FUNCTION_BLOCK FB_Cylinder_DualPWM_DualSensor EXTENDS FB_Cylinder_DualSensor
VAR_INPUT
END_VAR
VAR_OUTPUT
END_VAR
VAR
	fbPWMControl		: FB_Enfield_LSV_PWM_SolenoidControl;
	
	//Internal Property Values
	nDutyCycle		: INT := 100;
	
END_VAR

PROPERTY DutyCycle : INT
GET
DutyCycle := nDutyCycle;
END_GET
SET
nDutyCycle := DutyCycle;
END_SET
END_PROPERTY

METHOD HardwareUpdate : BOOL
VAR_INPUT
END_VAR
SUPER^.HardwareUpdate();

IF bExtendCommand THEN
	fbPWMControl.Actuate(nDutyCycle);
ELSIF bRetractCommand THEN
	fbPWMControl.Actuate(nDutyCycle * -1);
ELSE
	fbPWMControl.Actuate(0);
END_IF
END_METHOD

METHOD Monitoring : BOOL
VAR_INPUT
END_VAR
SUPER^.Monitoring();

bReady := bEnabled AND fbPWMControl.Ready AND NOT bError;
END_METHOD

END_FUNCTION_BLOCK

(* stored: Version 1.1.0.1, ProductVersion 3.1.4024.9
   POU FB_Cylinder_DualPWM_DualSensor: Id {b8f50960-2e92-4cf1-aa8b-435b0e5e3702}, SpecialFunc None
   Folder 01_SUPER_Overrides: Id {4a68cee4-2bb8-4c44-9106-a433d06ddca8}
   Property DutyCycle: Id {e5d3bd26-153e-42d6-92ff-5729a0f5e7e6}
   Get Get: Id {1da15d6b-cdec-49c0-bccf-2b889329b405}
   Set Set: Id {ab9e7f66-f68f-40d7-b2cd-22bd2ddac2b0}
   Method HardwareUpdate: Id {9cdcde0d-e8ec-4328-ba3d-a62092fdd57e}
   Method Monitoring: Id {0b748f5b-3920-48bb-a71d-ad8f3448fe53} *)
